Fanuc KAREL source: NC0008.KL

-- PROVISIONAL review KL for V770-1; original PC SHA256 57e1d8f6785279310a21831e8a997b45ff368435b6bd2584f347d57f169620fb
-- Incomplete behavior may be omitted. Consult companion uncertainty JSON. Do not deploy.
PROGRAM NC0008
%NOLOCKGROUP
-- UNRESOLVED_LOCAL_POOL 1 cells at code offset 3; source declarations unknown
-- DIRECT_LOCAL_WORD_ACCESS alone does not prove INTEGER, REAL, or BOOLEAN
BEGIN
  -- UNRESOLVED_PC offsets 0-8; opcodes 2B,2C,7B
  -- UNRESOLVED_PC offsets 13-20; opcodes 9D,23
  -- UNRESOLVED_PC offsets 25-38; opcodes 21,9D,57,79
  -- UNRESOLVED_PC offsets 43-56; opcodes 21,9D,57,79
  -- UNRESOLVED_PC offsets 61-74; opcodes 21,9D,57,79
  -- UNRESOLVED_PC offsets 79-92; opcodes 21,9D,57,79
  -- UNRESOLVED_PC offsets 97-110; opcodes 21,9D,57,79
  -- UNRESOLVED_PC offsets 115-128; opcodes 21,9D,57,79
  -- UNRESOLVED_PC offsets 133-146; opcodes 21,9D,57,79
  -- UNRESOLVED_PC offsets 151-164; opcodes 21,9D,57,79
  -- UNRESOLVED_PC offsets 169-182; opcodes 21,9D,57,79
  -- UNRESOLVED_PC offsets 187-200; opcodes 21,9D,57,79
  -- UNRESOLVED_PC offsets 205-218; opcodes 21,9D,57,79
  -- UNRESOLVED_PC offsets 223-236; opcodes 21,9D,57,79
  -- UNRESOLVED_PC offsets 241-255; opcodes 21,9D,52,23
  -- UNRESOLVED_PC offsets 260-265; opcodes 7A
  -- UNRESOLVED_PC offsets 270-288; opcodes 21,2E,52,23
  -- UNRESOLVED_PC offsets 298-303; opcodes 7A
  -- UNRESOLVED_PC offsets 308-326; opcodes 21,2E,52,23
  -- UNRESOLVED_PC offsets 336-341; opcodes 7A
  -- UNRESOLVED_PC offsets 346-364; opcodes 21,2E,52,23
  -- UNRESOLVED_PC offsets 374-379; opcodes 7A
  -- UNRESOLVED_PC offsets 384-402; opcodes 21,2E,52,23
  -- UNRESOLVED_PC offsets 412-417; opcodes 7A
  -- UNRESOLVED_PC offsets 422-440; opcodes 21,2E,52,23
  -- UNRESOLVED_PC offsets 450-455; opcodes 7A
  -- UNRESOLVED_PC offsets 460-478; opcodes 21,2E,52,23
  -- UNRESOLVED_PC offsets 488-493; opcodes 7A
  -- UNRESOLVED_PC offsets 498-516; opcodes 21,2E,52,23
  -- UNRESOLVED_PC offsets 526-531; opcodes 7A
  -- UNRESOLVED_PC offsets 536-554; opcodes 21,2E,52,23
  -- UNRESOLVED_PC offsets 564-569; opcodes 7A
  -- UNRESOLVED_PC offsets 574-592; opcodes 21,2E,52,23
  -- UNRESOLVED_PC offsets 602-607; opcodes 7A
  -- UNRESOLVED_PC offsets 612-630; opcodes 21,2E,52,23
  -- UNRESOLVED_PC offsets 640-645; opcodes 7A
  -- UNRESOLVED_PC offsets 650-668; opcodes 21,2E,52,23
  -- UNRESOLVED_PC offsets 678-683; opcodes 7A
  -- UNRESOLVED_PC offsets 688-706; opcodes 21,2E,52,23
  -- UNRESOLVED_PC offsets 716-720; opcodes 7F
  -- UNRESOLVED_PC offsets 725-729; opcodes 27,AA
  -- UNRESOLVED_PC offsets 734-738; opcodes 7F
END NC0008
